TYPE PLCopenRemoteInternal :
STRUCT
	Abort : BOOL;
	Status : PLCopenStatusBase;
END_STRUCT
END_TYPE

(* stored: Version 1.1.0.1
   DUT PLCopenRemoteInternal: Id {6734d06c-d81e-43fb-9b4f-7b69935b56e2} *)
